// TwinCAT 3 PLC project SVLS_MOT
// Title: SVLS MOTION
// Company: SLAC
// ProjectVersion: 0.0.0
// ProgramVersion: 3.1.4026.17
// libraries:
//   LCLS General, * (SLAC)
//   lcls-twincat-math, * (SLAC - LCLS)
//   lcls-twincat-motion, * (SLAC)
//   PMPS, * (SLAC - LCLS)
//   Tc2_MC2, * (Beckhoff Automation GmbH)
//   Tc2_Standard, * (Beckhoff Automation GmbH)
//   Tc2_System, * (Beckhoff Automation GmbH)
//   Tc2_Utilities, * (Beckhoff Automation GmbH)
//   Tc3_Module, * (Beckhoff Automation GmbH)
//   TcUnit, * (www.tcunit.org)
// project tree:
//   DUTs/ ST_EPSLimits.TcDUT (not stored)
//   GVLs/ Main.TcGVL (not stored)
//   ITFs/ I_ExternalSetpointGenerator.TcIO (not stored), I_HController.TcIO (not stored), I_CalculateHFromAngle.TcIO (not stored), I_MotionAxis.TcIO (not stored)
//   / PlcTask.TcTTO (not stored), ProductionPlcTask.TcTTO (not stored), TestPlcTask.TcTTO (not stored)
//   POUs/EPS/ FB_CheckEPS.TcPOU (not stored), FB_RestTimer.TcPOU (not stored), F_InRange.TcPOU (not stored), PRG_DET_Z_EPS.TcPOU (not stored)
//   POUs/FBs/ FB_ExternalSetpointGenerator.TcPOU (not stored), FB_HController.TcPOU (not stored), FB_CalculateHFromAngle.TcPOU (not stored), FB_MotionAxisNC.TcPOU (not stored)
//   POUs/ PRG_Main.TcPOU
//   Test/ FB_CalculateHFromAngle_Test.TcPOU (not stored), FB_HController_Test.TcPOU (not stored), FB_ExternalSetpointGenerator_Test.TcPOU (not stored), PRG_Test.TcPOU (not stored)
// real-time tasks:
//   TASK PlcTask: cycle T#10ms, priority 20, ADS port 350
//   TASK TestPlcTask: cycle T#10ms, priority 1, ADS port 351
//   TASK ProductionPlcTask: cycle T#10ms, priority 2, ADS port 352
// motion (NC):
// I/O:
//   DEVICE Device 1 (EtherCAT)
// variable links:
//   SVLS_MOT Instance <-> Device 1 (EtherCAT)/EK1200_01_00/EL5042_01_02-DET_Y-DET_Z
//     ProductionPlcTask Inputs/Main.M1.nRawEncoderULINT <-> FB Inputs Channel 1/Position
//     ProductionPlcTask Inputs/Main.M2.nRawEncoderULINT <-> FB Inputs Channel 2/Position
//   SVLS_MOT Instance <-> Device 1 (EtherCAT)/EK1200_01_00/EL5042_01_05-GRT_Y-SP5
//     ProductionPlcTask Inputs/Main.M3.nRawEncoderULINT <-> FB Inputs Channel 1/Position
//   SVLS_MOT Instance <-> Device 1 (EtherCAT)/EK1200_01_00/EL7047_01_01-DET_Y
//     ProductionPlcTask Inputs/Main.M1.bLimitBackwardEnable <-> STM Status/Status/Digital input 2
//     ProductionPlcTask Inputs/Main.M8.bLimitBackwardEnable <-> STM Status/Status/Digital input 2
//     ProductionPlcTask Inputs/Main.M1.bLimitForwardEnable <-> STM Status/Status/Digital input 1
//     ProductionPlcTask Inputs/Main.M8.bLimitForwardEnable <-> STM Status/Status/Digital input 1
//   SVLS_MOT Instance <-> Device 1 (EtherCAT)/EK1200_01_00/EL7047_01_03-DET_Z
//     ProductionPlcTask Inputs/Main.M2.bLimitBackwardEnable <-> STM Status/Status/Digital input 2
//     ProductionPlcTask Inputs/Main.M2.bLimitForwardEnable <-> STM Status/Status/Digital input 1
//   SVLS_MOT Instance <-> Device 1 (EtherCAT)/EK1200_01_00/EL7047_01_04-GRT_Y
//     ProductionPlcTask Inputs/Main.M3.bLimitBackwardEnable <-> STM Status/Status/Digital input 2
//     ProductionPlcTask Inputs/Main.M3.bLimitForwardEnable <-> STM Status/Status/Digital input 1
//   SVLS_MOT Instance <-> SVLS_MOTION SAF/Axes/ExternalSetpointGenerator_Test1
//     TestPlcTask Inputs/PRG_Test.AxisReference_ExternalSetpointGenerator_Test1.NcToPlc <-> Outputs/ToPlc
//     TestPlcTask Outputs/PRG_Test.AxisReference_ExternalSetpointGenerator_Test1.PlcToNc <-> Inputs/FromPlc
//   SVLS_MOT Instance <-> SVLS_MOTION SAF/Axes/ExternalSetpointGenerator_Test2
//     TestPlcTask Inputs/PRG_Test.AxisReference_ExternalSetpointGenerator_Test2.NcToPlc <-> Outputs/ToPlc
//     TestPlcTask Outputs/PRG_Test.AxisReference_ExternalSetpointGenerator_Test2.PlcToNc <-> Inputs/FromPlc
//   SVLS_MOT Instance <-> SVLS_MOTION SAF/Axes/HControllerDetAngle_Test1
//     TestPlcTask Inputs/PRG_Test.stMotionStage_HControllerDetAngle_Test1.Axis.NcToPlc <-> Outputs/ToPlc
//     TestPlcTask Outputs/PRG_Test.stMotionStage_HControllerDetAngle_Test1.Axis.PlcToNc <-> Inputs/FromPlc
//   SVLS_MOT Instance <-> SVLS_MOTION SAF/Axes/HControllerDetH_Test1
//     PlcTask Outputs/PRG_Test.fbHController_Test.nDetAngleEncoderComState_Test1 <-> Enc/Inputs/In/nComState
//     PlcTask Outputs/PRG_Test.fbHController_Test.nDetAngleEncoderState1_Test1 <-> Enc/Inputs/In/nState1
//     TestPlcTask Inputs/PRG_Test.stMotionStage_HControllerDetH_Test1.Axis.NcToPlc <-> Outputs/ToPlc
//     TestPlcTask Outputs/PRG_Test.stMotionStage_HControllerDetH_Test1.Axis.PlcToNc <-> Inputs/FromPlc
//   SVLS_MOT Instance <-> SVLS_MOTION SAF/Axes/M1_DET_Y_Angle
//     ProductionPlcTask Inputs/Main.M1.Axis.NcToPlc <-> Outputs/ToPlc
//     ProductionPlcTask Outputs/Main.M1.Axis.PlcToNc <-> Inputs/FromPlc
//   SVLS_MOT Instance <-> SVLS_MOTION SAF/Axes/M2_DET_Z
//     ProductionPlcTask Inputs/Main.M2.Axis.NcToPlc <-> Outputs/ToPlc
//     ProductionPlcTask Outputs/Main.M2.Axis.PlcToNc <-> Inputs/FromPlc
//   SVLS_MOT Instance <-> SVLS_MOTION SAF/Axes/M3_GRA_Y
//     ProductionPlcTask Inputs/Main.M3.Axis.NcToPlc <-> Outputs/ToPlc
//     ProductionPlcTask Outputs/Main.M3.Axis.PlcToNc <-> Inputs/FromPlc
//   SVLS_MOT Instance <-> SVLS_MOTION SAF/Axes/M8_Det_Y_H
//     ProductionPlcTask Inputs/Main.M8.Axis.NcToPlc <-> Outputs/ToPlc
//     ProductionPlcTask Outputs/Main.M8.Axis.PlcToNc <-> Inputs/FromPlc

// ---- POUs/PRG_Main.TcPOU

PROGRAM PRG_Main
VAR
    fbDetYAngle : FB_MotionStage;
    fbDetZ : FB_MotionStage;
    fbGraY : FB_MotionStage;
    fbDetYH : FB_MotionStage;
    bInit : BOOL := TRUE;

    fbMotionAxisDetAngle : FB_MotionAxisNC(
        AxisReference := Main.M1.Axis
    );
    fbMotionAxisDetH : FB_MotionAxisNC(
        AxisReference := Main.M8.Axis
    );
    fbCalculateHFromAngle : FB_CalculateHFromAngle(
        D_tu := 1238.29,
        R_a := 1200.10,
        R_c := 89.78
    );
    {attribute 'TcLinkTo' := '.nEncoderCount := TINC^SVLS_MOTION SAF^Axes^M8_Det_Y_H^Enc^Inputs^In^nDataIn1'}
    fbHController : FB_HController(
        iMotionAxisDetAngle := fbMotionAxisDetAngle,
        iCalculateHFromAngle := fbCalculateHFromAngle,
        stMotionStageAxisDetAngle := Main.M1,
        stMotionStageAxisDetH := Main.M8,
        bDetHMoveAbsoluteBusy := fbDetYH.fbDriveVirtual.fbMoveAbsolute.Busy
    );

END_VAR


IF bInit THEN
    bInit := FALSE;

    Main.M1.bHardwareEnable := TRUE;
    Main.M1.bPowerSelf := TRUE;
    Main.M1.nBrakeMode := ENUM_StageBrakeMode.NO_BRAKE;
    Main.M1.nEnableMode := ENUM_StageEnableMode.DURING_MOTION;

    Main.M2.bHardwareEnable := TRUE;
    Main.M2.bPowerSelf := TRUE;
    Main.M2.nBrakeMode := ENUM_StageBrakeMode.NO_BRAKE;
    Main.M2.nEnableMode := ENUM_StageEnableMode.DURING_MOTION;

    Main.M3.bHardwareEnable := TRUE;
    Main.M3.bPowerSelf := TRUE;
    Main.M3.nBrakeMode := ENUM_StageBrakeMode.NO_BRAKE;
    Main.M3.nEnableMode := ENUM_StageEnableMode.DURING_MOTION;

    Main.M8.bHardwareEnable := TRUE;
    Main.M8.bPowerSelf := TRUE;
    Main.M8.nBrakeMode := ENUM_StageBrakeMode.NO_BRAKE;
    Main.M8.nEnableMode := ENUM_StageEnableMode.DURING_MOTION;
END_IF

//PRG_DET_Z_EPS();

fbDetYAngle(stMotionStage:=Main.M1);
//fbHController();
fbDetYH(stMotionStage:=Main.M8);
fbDetZ(stMotionStage:=Main.M2);
fbGraY(stMotionStage:=Main.M3);

END_PROGRAM
